KUKA KRL data list: kuka_eki_hw_interface.dat

&ACCESS RVP
DEFDAT  KUKA_EKI_HW_INTERFACE
EXT  bas (BAS_COMMAND  :IN,REAL  :IN )
   ext bas(bas_command  :in,real  :in )
   INT id_count
ENDDAT
